Staubli VAL3: cycle_getList.pgx

program cycle_getList(num x_nType (dimensions=1))
  local num i
  local num nSize
  local string sName
begin
  //
  // Get the Cycle process list and put in the
  // global variable listProgram
  //
  // build the list
  nSize=size(listProgram)
  for i=1 to nSize-1
    delete(listProgram[0])
  endFor
  call cycle_getSize(nSize,x_nType)
  call cycle_getProg(sName,1,x_nType)
  // copy the list
  listProgram=sName
  if nSize>0
    for i=1 to nSize-1
      call cycle_getProg(sName,i+1,x_nType)
      insert(listProgram[i])
      listProgram[i]=sName
    endFor
  endIf
  //
end
